{attribute addProperty BoxType "EP7041-0002-0016"}
{attribute addProperty Id "StatusAT %I*Status_D6C17EA6445.51Counter_valueAT %I*UINT16217Latch_valueAT %I*UINT16218"}
{attribute addProperty CRC "592369733"}
{attribute addProperty SizeInBites "76"}
{attribute addProperty SizeInBytes "9.5"}
TYPE ENC_Status_compact_234ED845 :
STRUCT
	{attribute addProperty Name "Status"}
	Status AT %I* : Status_D6C17EA6;
	{attribute addProperty Name "Counter_value"}
	Counter_value AT %I* : UINT;
	{attribute addProperty Name "Latch_value"}
	Latch_value AT %I* : UINT;
END_STRUCT
END_TYPE

(* stored: Version 1.2.0.0, ProductVersion 3.1.4024.9
   DUT ENC_Status_compact_234ED845: Id {65381ca7-e6b9-46ae-95ce-810a3968cc2f} *)
